(* IEC 61131-3 sources: tuk_project/src/control_systems/implementation/editor/Sensor+PusherTest/build, 2 files *)

(* ---- plc.st ---- *)
TYPE
  LOGLEVEL : (CRITICAL, WARNING, INFO, DEBUG) := INFO;
END_TYPE

FUNCTION_BLOCK LOGGER
  VAR_INPUT
    TRIG : BOOL;
    MSG : STRING;
    LEVEL : LOGLEVEL := INFO;
  END_VAR
  VAR
    TRIG0 : BOOL;
  END_VAR

  IF TRIG AND NOT TRIG0 THEN
  {{
   LogMessage(GetFbVar(LEVEL),(char*)GetFbVar(MSG, .body),GetFbVar(MSG, .len));
  }}
  END_IF;
  TRIG0:=TRIG;
END_FUNCTION_BLOCK

FUNCTION_BLOCK python_eval
  VAR_INPUT
    TRIG : BOOL;
    CODE : STRING;
  END_VAR
  VAR_OUTPUT
    ACK : BOOL;
    RESULT : STRING;
  END_VAR
  VAR
    STATE : DWORD;
    BUFFER : STRING;
    PREBUFFER : STRING;
    TRIGM1 : BOOL;
    TRIGGED : BOOL;
  END_VAR

  {extern void __PythonEvalFB(int, PYTHON_EVAL*);__PythonEvalFB(0, data__);}
END_FUNCTION_BLOCK

FUNCTION_BLOCK python_poll
  VAR_INPUT
    TRIG : BOOL;
    CODE : STRING;
  END_VAR
  VAR_OUTPUT
    ACK : BOOL;
    RESULT : STRING;
  END_VAR
  VAR
    STATE : DWORD;
    BUFFER : STRING;
    PREBUFFER : STRING;
    TRIGM1 : BOOL;
    TRIGGED : BOOL;
  END_VAR

  {extern void __PythonEvalFB(int, PYTHON_EVAL*);__PythonEvalFB(1,(PYTHON_EVAL*)(void*)data__);}
END_FUNCTION_BLOCK

FUNCTION_BLOCK python_gear
  VAR_INPUT
    N : UINT;
    TRIG : BOOL;
    CODE : STRING;
  END_VAR
  VAR_OUTPUT
    ACK : BOOL;
    RESULT : STRING;
  END_VAR
  VAR
    py_eval : python_eval;
    COUNTER : UINT;
    ADD10_OUT : UINT;
    EQ13_OUT : BOOL;
    SEL15_OUT : UINT;
    AND7_OUT : BOOL;
  END_VAR

  ADD10_OUT := ADD(COUNTER, 1);
  EQ13_OUT := EQ(N, ADD10_OUT);
  SEL15_OUT := SEL(EQ13_OUT, ADD10_OUT, 0);
  COUNTER := SEL15_OUT;
  AND7_OUT := AND(EQ13_OUT, TRIG);
  py_eval(TRIG := AND7_OUT, CODE := CODE);
  ACK := py_eval.ACK;
  RESULT := py_eval.RESULT;
END_FUNCTION_BLOCK

PROGRAM program0
  VAR
    Sensor : BOOL;
    PusherFront : BOOL;
    Reset : BOOL;
    Pusher : BOOL := 0;
    InConveyor : BOOL := 1;
    OutConveyor : BOOL := 1;
  END_VAR
  VAR
    T1 : TON;
    Temp : BOOL := 0;
  END_VAR

  T1(IN:=Temp, PT:= T#2000ms);

  IF Reset THEN

    Pusher:= 0;
    Temp:= 0;

  END_IF;

  IF Sensor THEN

    Temp:= 1;

  END_IF;

  IF T1.Q THEN

    Pusher:= 1;
    Temp:=0;

  END_IF;

  IF PusherFront THEN

    Pusher:= 0;

  END_IF;

END_PROGRAM

CONFIGURATION Config0

  RESOURCE Res0 ON PLC
    TASK task0(INTERVAL := T#20ms,PRIORITY := 0);
    PROGRAM instance0 WITH task0 : program0;
  END_RESOURCE
END_CONFIGURATION

(* ---- generated_plc.st ---- *)
PROGRAM program0
  VAR
    Sensor AT %IX100.0 : BOOL;
    PusherFront AT %IX100.1 : BOOL;
    Reset AT %IX100.7 : BOOL;
    Pusher AT %QX100.1 : BOOL := 0;
    InConveyor AT %QX100.0 : BOOL := 1;
    OutConveyor AT %QX100.2 : BOOL := 1;
  END_VAR
  VAR
    T1 : TON;
    Temp : BOOL := 0;
  END_VAR

  T1(IN:=Temp, PT:= T#2000ms);

  IF Reset THEN

    Pusher:= 0;
    Temp:= 0;

  END_IF;

  IF Sensor THEN

    Temp:= 1;

  END_IF;

  IF T1.Q THEN

    Pusher:= 1;
    Temp:=0;

  END_IF;

  IF PusherFront THEN

    Pusher:= 0;

  END_IF;

END_PROGRAM

CONFIGURATION Config0

  RESOURCE Res0 ON PLC
    TASK task0(INTERVAL := T#20ms,PRIORITY := 0);
    PROGRAM instance0 WITH task0 : program0;
  END_RESOURCE
END_CONFIGURATION
